FUNCTION_BLOCK FB_LaudaResponse
VAR_INPUT
	sResponse	: Tc2_System.T_MaxString;
END_VAR
VAR_OUTPUT
END_VAR
VAR
END_VAR

PROPERTY PUBLIC RawValue : T_MaxString
GET
RawValue := sResponse;
END_GET
END_PROPERTY

PROPERTY PUBLIC Success : BOOL
GET
Success := 
	LaudaHelper.ValidateReadCommandResponse(sResponse) AND 
	LaudaHelper.ValidateSendCommandResponse(sResponse);
END_GET
END_PROPERTY

PROPERTY PUBLIC WithoutSuffix : T_MaxString
GET
WithoutSuffix := LaudaHelper.RemoveSuffix(sResponse);
END_GET
END_PROPERTY

END_FUNCTION_BLOCK

(* stored: Version 1.1.0.1, ProductVersion 3.1.4024.12
   POU FB_LaudaResponse: Id {35f8e709-f468-0b47-138a-bcaf5861f7b3}, SpecialFunc None
   Property RawValue: Id {83553254-5c35-0f94-3c3d-643eb9abc761}
   Get Get: Id {f6c1035a-83f6-0315-27aa-65c620878c7a}
   Property Success: Id {8504984e-2e04-02a7-3338-8921ffa3e826}
   Get Get: Id {2e981743-ad83-0198-2b09-8d166c464498}
   Property WithoutSuffix: Id {5db934a5-bf0e-0460-0850-ac7dc3d38e78}
   Get Get: Id {f56c6fe2-fca1-0d67-02b1-fe7db726cfdf} *)
